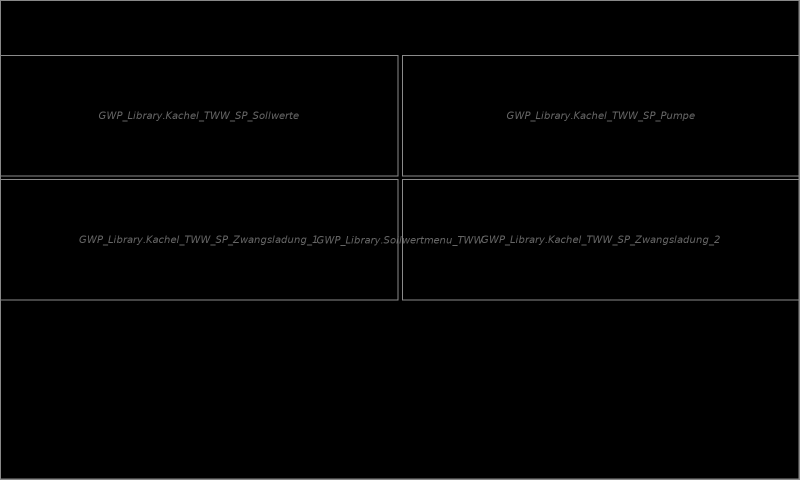
VISUALIZATION Sollwertmenu_TWW  // 800x480
    Frame (0,0 800x480)
        shows GWP_Library.Sollwertmenu_TWW(FB_Init_1 := Main.Init_0)
    Frame (0,55 398x121)
        shows GWP_Library.Kachel_TWW_SP_Sollwerte()
        OnMouseClick: change screen: TWW_SP_Sollwerte
    Frame (402,55 398x121)
        shows GWP_Library.Kachel_TWW_SP_Pumpe()
        OnMouseClick: change screen: TWW_SP_PU_Sollwerte
    Frame (0,179 398x121)
        shows GWP_Library.Kachel_TWW_SP_Zwangsladung_1()
        OnMouseClick: change screen: TWW_SP_CLK_I_Zwangsladung_1
    Frame (402,179 398x121)
        shows GWP_Library.Kachel_TWW_SP_Zwangsladung_2()
        OnMouseClick: change screen: TWW_SP_CLK_I_Zwangsladung_2
END_VISUALIZATION

(* stored: Version 1.1.0.1, ProductVersion 3.1.4022.6
   Visu Sollwertmenu_TWW: Id {0775b5a5-6f1c-40a3-b655-d558b7960656} *)
